PROGRAM MAIN
VAR
END_VAR

IF Inputs.bEnableSimulation THEN
	CraneSimulation();
END_IF;

END_PROGRAM

(* stored: Version 1.1.0.1, ProductVersion 3.1.4024.10
   POU MAIN: Id {ac89f347-c6c6-419e-a490-7d92bdd5a582}, SpecialFunc None *)
